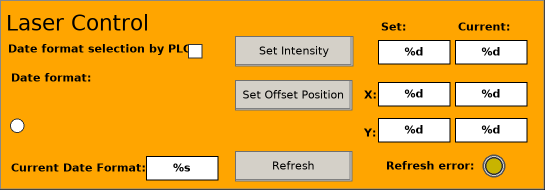
VISUALIZATION vLaserControl_old  // 545x190
VAR_IN_OUT
	stHMI: stHMI_Laser;
END_VAR
    Rectangle (0,0 545x190)
    RadioButton (8,92 150x67), variable: stHMI.iSelectMarking, input disabled if: GVL.fbUserLogin.nUserRole <> nSQL_UserRoles.Maintenance
        Areas[0]: Text=Year - Week
        Areas[1]: Text=Year - Month
    Label (5,37 226x24), "Date format selection by PLC"
    Label (9,63 226x24)
    Label (8,66 226x24), "Date format:"
    Checkbox (186,38 26x26), variable: stHMI.bEnableLaserTCPCOmmunication, input disabled if: GVL.fbUserLogin.nUserRole <> nSQL_UserRoles.Maintenance
    Label (8,156 226x24), "Current Date Format:"
    Rectangle (146,156 72x24), "%s", text variable: stHMI.sCurrentDateText, input disabled if: TRUE
    Button (235,36 118x30), "Set Intensity", colour toggle: stHMI.bSetIntensityOK, input disabled if: GVL.fbUserLogin.nUserRole <> nSQL_UserRoles.Maintenance
        OnMouseDown: execute { stHMI.bReqSetIntensity :=TRUE; }
    Button (235,80 117x30), "Set Offset Position", colour toggle: stHMI.bSetPositionOK, input disabled if: GVL.fbUserLogin.nUserRole <> nSQL_UserRoles.Maintenance
        OnMouseDown: execute { stHMI.bReqSetPosition:=TRUE; }
    Rectangle (378,40 72x24), "%d", text variable: stHMI.iIntensity_OUT, input disabled if: GVL.fbUserLogin.nUserRole <> nSQL_UserRoles.Maintenance
        OnMouseDown: write the text variable via VisuDialogs.Numpad, min 0, max 100
    Rectangle (378,82 72x24), "%d", text variable: stHMI.iPositionX_OUT, input disabled if: GVL.fbUserLogin.nUserRole <> nSQL_UserRoles.Maintenance
        OnMouseDown: write the text variable via VisuDialogs.Numpad, min 0
    Rectangle (378,118 72x24), "%d", text variable: stHMI.iPositionY_OUT, input disabled if: GVL.fbUserLogin.nUserRole <> nSQL_UserRoles.Maintenance
        OnMouseDown: write the text variable via VisuDialogs.Numpad, min 0
    Label (361,83 24x24), "X:"
    Label (361,121 24x24), "Y:"
    Rectangle (455,40 72x24), "%d", text variable: stHMI.iIntensity_IN, input disabled if: TRUE
    Rectangle (455,82 72x24), "%d", text variable: stHMI.iPositionX_IN, input disabled if: TRUE
    Rectangle (455,118 72x24), "%d", text variable: stHMI.iPositionY_IN, input disabled if: TRUE
    Label (378,15 55x24), "Set:"
    Label (455,15 55x24), "Current:"
    Button (235,151 117x30), "Refresh", input disabled if: GVL.fbUserLogin.nUserRole <> nSQL_UserRoles.Maintenance
        OnMouseDown: execute { stHMI.bReqRefreshParams:=TRUE; }
    Lamp1 (481,153 26x26), variable: stHMI.bRefreshError, style: Lamp-Lamp1-Yellow
    Label (383,154 87x24), "Refresh error:"
    Label (3,8 156x30), "Laser Control"
END_VISUALIZATION

(* stored: Version 1.1.0.1, ProductVersion 3.1.4024.15
   Visu vLaserControl_old: Id {977b251f-40ec-42d7-aa21-096aef2ec150} *)
